{attribute 'qualified_only'}
{attribute 'strict'}
TYPE E_ModbusDataType :
(
	uint16,
	uint32,
	uint64
);
END_TYPE

(* stored: Version 1.1.0.1, ProductVersion 3.1.4024.12
   DUT E_ModbusDataType: Id {3876068c-9938-4252-8736-fc9a7d2498a3} *)
